TYPE ST_RobotLineBox_HWI :
STRUCT
  stInN01_1008State       : ST_CardState_HWI;//CGSMini_Robot01LineBoxInN01-EL1008
  stAnaInN01_3202State    : ST_CardState_HWI;//CGSMini_Robot01LineBoxAnaInN01-EL3202
  stAnaInN02_3054State    : ST_CardState_HWI;//CGSMini_Robot01LineBoxAnaInN02-EL3054
  stAnaInN03_3202State    : ST_CardState_HWI;//CGSMini_Robot01LineBoxAnaInN03-EL3202
  stOverCProt1_9222State  : ST_CardState_HWI;//CGSMini_Robot01LineBoxOverCurrProt1-EL9222
  stLineBox_1100State     : ST_CardState_HWI;//CGSMini_Robot01LineBoxBox-EK1100 not yet available useful in case of only one PLC for all robots line
  stSafety_1918State      : ST_CardState_HWI;//CGSMini_Robot01LineBoxSafeInN01-EL1918
 
  stRobotID               : ST_RobotIdentification_HWI;//CGSMini_Robot01LineBoxInN01-EL1008
  stRemoteCtrl            : ST_RemoteControl_HWI;//CGSMini_Robot01LineBoxInN01-EL1008
  stOverCProt             : ST_OverCurrProtection_HWI;//CGSMini_Robot01LineBoxOverCurrProt1-EL9222
  stAnaRTDLine1           : ST_Analog_HWI;//CGSMini_Robot01LineBoxAnaInN01-EL3202 RTD1
  stAnaRTDLine2           : ST_Analog_HWI;//CGSMini_Robot01LineBoxAnaInN01-EL3202 RTD2
	stAnaFlowLine1          : ST_Analog_HWI;//CGSMini_Robot01LineBoxAnaInN02-EL3054 
  stAnaFlowLine2          : ST_Analog_HWI;//CGSMini_Robot01LineBoxAnaInN02-EL3054 
  stAnaPressure           : ST_Analog_HWI;//CGSMini_Robot01LineBoxAnaInN02-EL3054
  stAnaRTDInternal        : ST_Analog_HWI;//CGSMini_Robot01LineBoxAnaInN03-EL3202 RTDInternal
  stAnaRTDExternal        : ST_Analog_HWI;//CGSMini_Robot01LineBoxAnaInN03-EL3202 RTDExternal
END_STRUCT
END_TYPE

(* stored: Version 1.1.0.1, ProductVersion 3.1.4024.12
   DUT ST_RobotLineBox_HWI: Id {0919acf6-4c6c-4180-a98b-89bf315404db} *)
